// Mitsubishi GX Works2 project: LRI - Lógica NOR   PLC: Q03UDV
// HelloWorld

PROGRAM MAIN
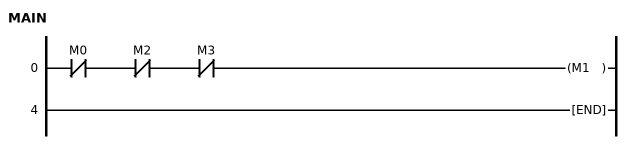
0     LDI     M0
      ANI     M2
      ANI     M3
      OUT     M1
4     END
END_PROGRAM
